PROGRAM SimutateHwModules
VAR
	stHardwareId : ST_HardwareId;
END_VAR

fbXDriveBeck.P_pMultiZRef := ADR(aFbMultiZRef[1]);
fbYDriveBeck.P_pMultiZRef := ADR(aFbMultiZRef[1]);
stHardwareId.eGroup := E_HardwareGrp.AxisX;
stHardwareId.nParentItem := 0;
stHardwareId.nItem := 1;
fbXDriveBeck.P_stHardwareId := stHardwareId;
stHardwareId.eGroup := E_HardwareGrp.AxisY;
stHardwareId.nParentItem := 1;
stHardwareId.nItem := 1;
fbYDriveBeck.P_stHardwareId := stHardwareId;
 
fbXYDriveList.M_Add(ADR(fbXDriveBeck));
fbXYDriveList.M_Add(ADR(fbYDriveBeck));

END_PROGRAM

(* stored: Version 1.1.0.1, ProductVersion 3.1.4020.12
   POU SimutateHwModules: Id {dc8ef37f-0f03-4e8a-9c29-20627da88774}, SpecialFunc None *)
